// TIA Portal V17 program export: 1 tag tables, 0 data types, 0 data blocks, 3 code blocks (in call order from the OBs), 1 instance data blocks

VAR_GLOBAL   // PLC tag table "Default tag table_2"
END_VAR
VAR_GLOBAL CONSTANT   // user constants
   MAXTIME : Time := T#6s;
END_VAR

ORGANIZATION_BLOCK "MainConveyor"   // OB1, LAD, ProgramCycle
TITLE = "Main Program Sweep (Cycle)"
VERSION : 0.1
// stored: AutoNumber true, IsIECCheckEnabled false, SetENOAutomatically false
   VAR_INPUT
      Initial_Call : Bool;   // Initial call of this OB
      Remanence : Bool;   // =True, if remanent data are available
   END_VAR
BEGIN

REGION Network 1
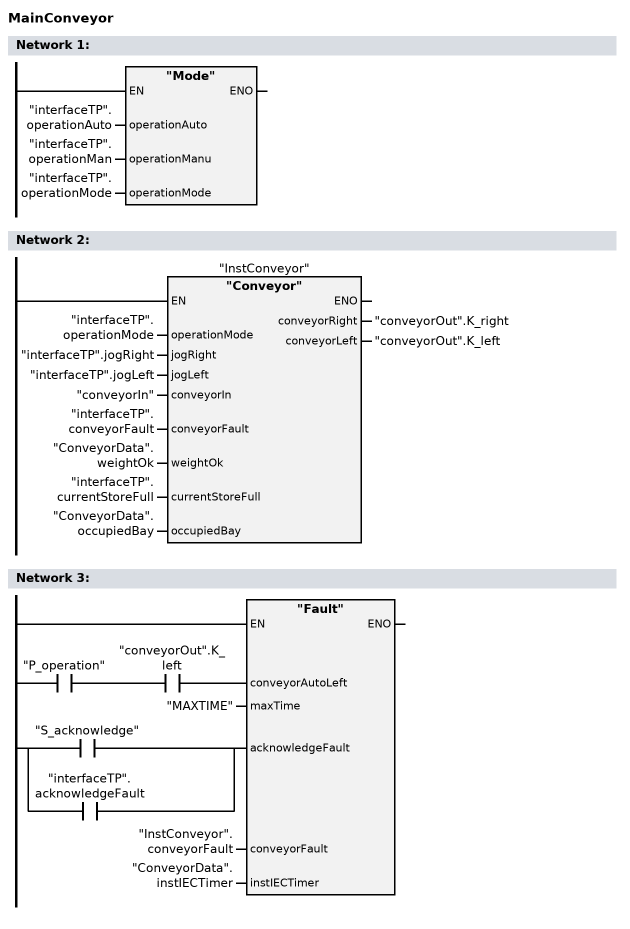
   RUNG wire#powerrail
      "Mode"(operationAuto := "interfaceTP".operationAuto, operationManu := "interfaceTP".operationMan, operationMode := "interfaceTP".operationMode)
   END_RUNG
   // the same network as SCL:
   "Mode"(operationAuto := "interfaceTP".operationAuto,
          operationManu := "interfaceTP".operationMan,
          operationMode := "interfaceTP".operationMode);
END_REGION

REGION Network 2
   RUNG wire#powerrail
      "InstConveyor"(operationMode := "interfaceTP".operationMode, jogRight := "interfaceTP".jogRight, jogLeft := "interfaceTP".jogLeft, conveyorIn := "conveyorIn", conveyorFault := "interfaceTP".conveyorFault, weightOk := "ConveyorData".weightOk, currentStoreFull := "interfaceTP".currentStoreFull, occupiedBay := "ConveyorData".occupiedBay, conveyorRight => "conveyorOut".K_right, conveyorLeft => "conveyorOut".K_left)
   END_RUNG
   // the same network as SCL:
   "InstConveyor"(operationMode := "interfaceTP".operationMode,   // "Conveyor"
                  jogRight := "interfaceTP".jogRight,
                  jogLeft := "interfaceTP".jogLeft,
                  conveyorIn := "conveyorIn",
                  conveyorFault := "interfaceTP".conveyorFault,
                  weightOk := "ConveyorData".weightOk,
                  currentStoreFull := "interfaceTP".currentStoreFull,
                  occupiedBay := "ConveyorData".occupiedBay,
                  conveyorRight => "conveyorOut".K_right,
                  conveyorLeft => "conveyorOut".K_left);
END_REGION

REGION Network 3
   RUNG wire#powerrail
      "Fault"(conveyorAutoLeft := wire#w1, acknowledgeFault := wire#w2, maxTime := "MAXTIME", conveyorFault := "InstConveyor".conveyorFault, instIECTimer := "ConveyorData".instIECTimer)
   END_RUNG
   RUNG wire#powerrail
      Contact( "P_operation" )
      Contact( "conveyorOut".K_left )
   END_RUNG wire#w1
   RUNG wire#powerrail
      Contact( "S_acknowledge" )
   END_RUNG wire#w2
   RUNG wire#powerrail
      Contact( "interfaceTP".acknowledgeFault )
   END_RUNG wire#w2
   // the same network as SCL:
   "Fault"(conveyorAutoLeft := "P_operation" AND "conveyorOut".K_left,
           maxTime := "MAXTIME",
           acknowledgeFault := "S_acknowledge" OR "interfaceTP".acknowledgeFault,
           conveyorFault := "InstConveyor".conveyorFault,
           instIECTimer := "ConveyorData".instIECTimer);
END_REGION
END_ORGANIZATION_BLOCK

FUNCTION_BLOCK "Conveyor"   // FB2, LAD
VERSION : 0.1
// stored: Access Published, AutoNumber true, IsIECCheckEnabled false, IsRetainMemResEnabled false, MemoryReserve 100, SetENOAutomatically false, UDAEnableTagReadback false
   VAR_INPUT
      operationMode : Bool;
      jogRight : Bool;
      jogLeft : Bool;
      conveyorIn : "typeConveyorInput";
      conveyorFault : Bool;
      weightOk : Bool;
      currentStoreFull : Bool;
   END_VAR
   VAR_OUTPUT
      conveyorRight : Bool;
      conveyorLeft : Bool;
   END_VAR
   VAR_IN_OUT
      occupiedBay : Array[#FIRSTBAY..#LASTBAY] of Bool;
   END_VAR
   VAR
      statAutoLeft : Bool;
      InstBayOccupied1 { S7_SetPoint := 'True'} : "BayOccupied";
      InstBayOccupied2 { S7_SetPoint := 'True'} : "BayOccupied";
      InstBayOccupied3 { S7_SetPoint := 'True'} : "BayOccupied";
   END_VAR
   VAR_TEMP
      tempManLeft : Bool;
   END_VAR
   VAR CONSTANT
      FIRSTBAY : UInt := 1;
      LASTBAY : UInt := 3;
   END_VAR
BEGIN

REGION Network 1
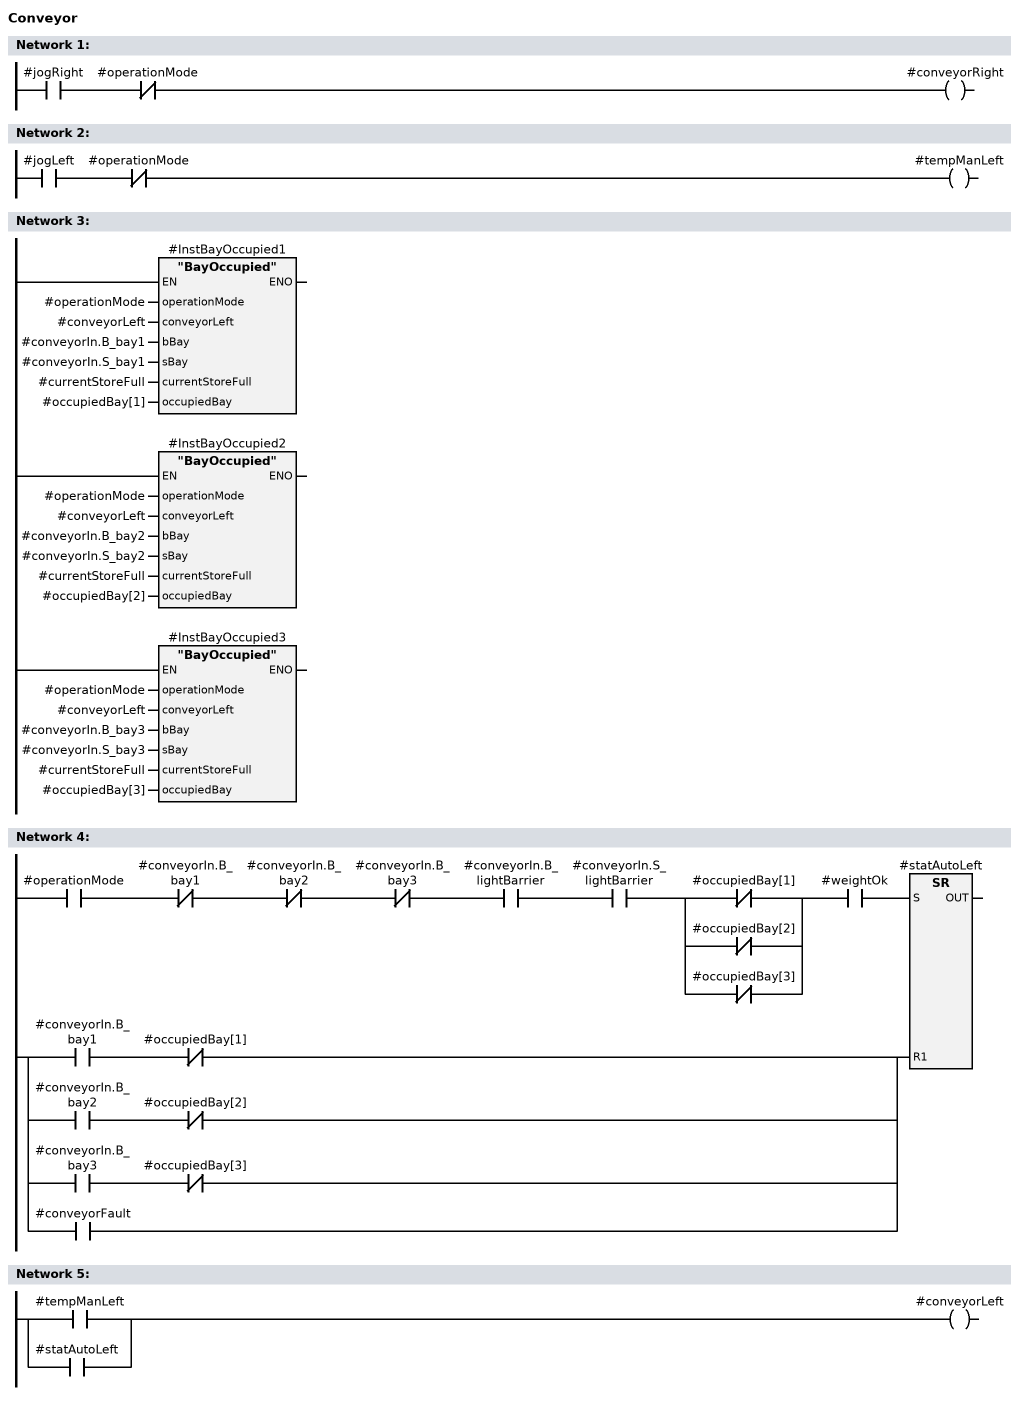
   RUNG wire#powerrail
      Contact( #jogRight )
      I_Contact( #operationMode )
      Coil( #conveyorRight )
   END_RUNG
   // the same network as SCL:
   #conveyorRight := #jogRight AND NOT #operationMode;
END_REGION

REGION Network 2
   RUNG wire#powerrail
      Contact( #jogLeft )
      I_Contact( #operationMode )
      Coil( #tempManLeft )
   END_RUNG
   // the same network as SCL:
   #tempManLeft := #jogLeft AND NOT #operationMode;
END_REGION

REGION Network 3
   RUNG wire#powerrail
      #InstBayOccupied1(operationMode := #operationMode, conveyorLeft := #conveyorLeft, bBay := #conveyorIn.B_bay1, sBay := #conveyorIn.S_bay1, currentStoreFull := #currentStoreFull, occupiedBay := #occupiedBay[1])
   END_RUNG
   RUNG wire#powerrail
      #InstBayOccupied2(operationMode := #operationMode, conveyorLeft := #conveyorLeft, bBay := #conveyorIn.B_bay2, sBay := #conveyorIn.S_bay2, currentStoreFull := #currentStoreFull, occupiedBay := #occupiedBay[2])
   END_RUNG
   RUNG wire#powerrail
      #InstBayOccupied3(operationMode := #operationMode, conveyorLeft := #conveyorLeft, bBay := #conveyorIn.B_bay3, sBay := #conveyorIn.S_bay3, currentStoreFull := #currentStoreFull, occupiedBay := #occupiedBay[3])
   END_RUNG
   // the same network as SCL:
   #InstBayOccupied1(operationMode := #operationMode,   // "BayOccupied"
                     conveyorLeft := #conveyorLeft,
                     bBay := #conveyorIn.B_bay1,
                     sBay := #conveyorIn.S_bay1,
                     currentStoreFull := #currentStoreFull,
                     occupiedBay := #occupiedBay[1]);
   #InstBayOccupied2(operationMode := #operationMode,   // "BayOccupied"
                     conveyorLeft := #conveyorLeft,
                     bBay := #conveyorIn.B_bay2,
                     sBay := #conveyorIn.S_bay2,
                     currentStoreFull := #currentStoreFull,
                     occupiedBay := #occupiedBay[2]);
   #InstBayOccupied3(operationMode := #operationMode,   // "BayOccupied"
                     conveyorLeft := #conveyorLeft,
                     bBay := #conveyorIn.B_bay3,
                     sBay := #conveyorIn.S_bay3,
                     currentStoreFull := #currentStoreFull,
                     occupiedBay := #occupiedBay[3]);
END_REGION

REGION Network 4
   RUNG wire#powerrail
      Contact( #operationMode )
      I_Contact( #conveyorIn.B_bay1 )
      I_Contact( #conveyorIn.B_bay2 )
      I_Contact( #conveyorIn.B_bay3 )
      Contact( #conveyorIn.B_lightBarrier )
      Contact( #conveyorIn.S_lightBarrier )
      wire#w1
      I_Contact( #occupiedBay[1] )
      wire#w2
      Contact( #weightOk )
      S_SR(operand := #statAutoLeft, r1 := wire#w3)
   END_RUNG
   RUNG wire#w1
      I_Contact( #occupiedBay[2] )
   END_RUNG wire#w2
   RUNG wire#w1
      I_Contact( #occupiedBay[3] )
   END_RUNG wire#w2
   RUNG wire#powerrail
      Contact( #conveyorIn.B_bay1 )
      I_Contact( #occupiedBay[1] )
   END_RUNG wire#w3
   RUNG wire#powerrail
      Contact( #conveyorIn.B_bay2 )
      I_Contact( #occupiedBay[2] )
   END_RUNG wire#w3
   RUNG wire#powerrail
      Contact( #conveyorIn.B_bay3 )
      I_Contact( #occupiedBay[3] )
   END_RUNG wire#w3
   RUNG wire#powerrail
      Contact( #conveyorFault )
   END_RUNG wire#w3
   // the same network as SCL:
   IF #operationMode AND NOT #conveyorIn.B_bay1 AND NOT #conveyorIn.B_bay2 AND NOT #conveyorIn.B_bay3 AND #conveyorIn.B_lightBarrier AND #conveyorIn.S_lightBarrier AND (NOT #occupiedBay[1] OR NOT #occupiedBay[2] OR NOT #occupiedBay[3]) AND #weightOk THEN
       #statAutoLeft := TRUE;   // SR flip-flop
   END_IF;
   IF (#conveyorIn.B_bay1 AND NOT #occupiedBay[1]) OR (#conveyorIn.B_bay2 AND NOT #occupiedBay[2]) OR (#conveyorIn.B_bay3 AND NOT #occupiedBay[3]) OR #conveyorFault THEN
       #statAutoLeft := FALSE;
   END_IF;
END_REGION

REGION Network 5
   RUNG wire#powerrail
      Contact( #tempManLeft )
      wire#w1
      Coil( #conveyorLeft )
   END_RUNG
   RUNG wire#powerrail
      Contact( #statAutoLeft )
   END_RUNG wire#w1
   // the same network as SCL:
   #conveyorLeft := #tempManLeft OR #statAutoLeft;
END_REGION
END_FUNCTION_BLOCK

FUNCTION_BLOCK "BayOccupied"   // FB3, LAD
VERSION : 0.1
// stored: Access Published, AutoNumber true, IsIECCheckEnabled false, IsRetainMemResEnabled false, MemoryReserve 100, SetENOAutomatically false, UDAEnableTagReadback false
   VAR_INPUT
      operationMode : Bool;
      conveyorLeft : Bool;
      bBay : Bool;
      sBay : Bool;
      currentStoreFull : Bool;
   END_VAR
   VAR_IN_OUT
      occupiedBay : Bool;
   END_VAR
   VAR
      staOldConveyorLeft : Bool;
   END_VAR
   VAR_TEMP   // added for the SCL form of the ladder/FBD networks
      _w1 : Bool;
      _w2 : Bool;
   END_VAR
BEGIN

REGION Network 1
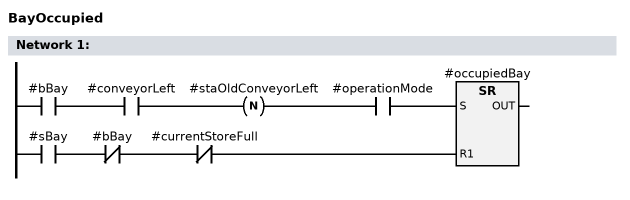
   RUNG wire#powerrail
      Contact( #bBay )
      Contact( #conveyorLeft )
      N_Trig( #staOldConveyorLeft )
      Contact( #operationMode )
      S_SR(operand := #occupiedBay, r1 := wire#w1)
   END_RUNG
   RUNG wire#powerrail
      Contact( #sBay )
      I_Contact( #bBay )
      I_Contact( #currentStoreFull )
   END_RUNG wire#w1
   // the same network as SCL:
   #_w1 := #bBay AND #conveyorLeft;
   #_w2 := NOT #_w1 AND #staOldConveyorLeft;   // falling edge
   #staOldConveyorLeft := #_w1;
   IF #_w2 AND #operationMode THEN
       #occupiedBay := TRUE;   // SR flip-flop
   END_IF;
   IF #sBay AND NOT #bBay AND NOT #currentStoreFull THEN #occupiedBay := FALSE; END_IF;
END_REGION
END_FUNCTION_BLOCK

DATA_BLOCK "InstConveyor"   // DB4
VERSION : 0.1
// stored: Access Unpublished, AutoNumber true, DBAccessibleFromOPCUA true, DBAccessibleFromWebserver true, InstanceOfName Conveyor, InstanceOfType FB
"Conveyor"
BEGIN
END_DATA_BLOCK
